TYPE ST_APP_CTRL :
STRUCT
  Cmd       : E_INSTANCE_CMD;
  Variant   : E_APP_VARIANT;
END_STRUCT
END_TYPE

(* stored: Version 1.1.0.1
   DUT ST_APP_CTRL: Id {18c7c16c-1097-4c1b-8405-47d2cee4cf30} *)
